{attribute 'pack_mode' := '1'}
TYPE ST_AdsSettingsBatch :
	STRUCT
		nMagic : UDINT := 16#41534554;       // "ASET"
		nFormatVersion : UINT := 2;
		nPayloadSize : UINT := 184;
		nSequenceStart : UDINT := 0;
		nRequestId : UDINT := 0;
		nAxisMask : BYTE := 0;
		nReservedByte : BYTE := 0;
		nReserved : UINT := 0;
		stAxisX : ST_Settings;
		stAxisY : ST_Settings;
		nSequenceEnd : UDINT := 0;
	END_STRUCT
END_TYPE

(* stored: Version 1.1.0.1, ProductVersion 3.1.4024.15
   DUT ST_AdsSettingsBatch: Id {d284e246-3f91-45c5-9da9-1f097f49e85f} *)
